// TIA Portal V21 export
TYPE "LBC_Basic_typeAnalogOutputInterface"
TITLE = LBC_typeAnalogOutputInterface_Basic
// Module interface for external systems
   STRUCT
      commands : "LBC_typeInterfaceCommands";
      monitoring { ExternalWritable := 'False'} : "LBC_typeAnalogProcessValues_Basic";
      configuration : "LBC_typeAnalogOutputConfiguration_Basic";
   END_STRUCT;
END_TYPE
